FUNCTION_BLOCK Test_F_DateTimeAsString_ms EXTENDS T_UnitTestBase
VAR
    TimeStruct : TIMESTRUCT := (wDay          := 23,
                                wMonth        := 12,
                                wYear         := 1945,
                                wHour         := 22,
                                wMinute       := 20,
                                wSecond       := 18,
                                wMilliseconds := 512);
END_VAR

METHOD Init
VAR_INPUT
END_VAR
END_METHOD

{attribute 'analysis' := '-33'} // inhibit unused variable warning
METHOD RunTest
AssertEquals_STRING(Expected := '22:20:18.512 23/12/1945',
                    Actual   := F_DateTimeAsString_ms(TimeStruct),
                    Message  := 'F_DateTimeAsString_ms(TimeStruct)');

TestCompleted := TRUE;
END_METHOD

END_FUNCTION_BLOCK

(* stored: Version 1.1.0.1, ProductVersion 3.1.4024.12
   POU Test_F_DateTimeAsString_ms: Id {3b9edf74-0e2a-0b80-276d-9d87de77dccc}, SpecialFunc None
   Method Init: Id {6c13043b-7332-055c-3ef0-53f72d746232}
   Method RunTest: Id {f3715779-e847-0e84-1f69-8e9ca4a7dbed} *)
